(*
		The sequence manager co-ordinates the selection and execution of 
		machine sequences. Machine sequences are created by extending the 
		FB_SequenceBase FB.
*)
FUNCTION_BLOCK FB_SequenceManager_ss
VAR	
	//aSequences: ARRAY[1..5] OF POINTER TO FB_SequenceBase;
	 
	nNumberSequences: INT := 0;
	
	{attribute 'OPC.UA.DA' := '1'} 
	eState:  E_SequenceState := E_SequenceState.STOP; //always stop sequences after PLC restart
	{attribute 'OPC.UA.DA' := '1'} 
	eStateTarget:  E_SequenceState := E_SequenceState.STOP;
	
	eSMState: (STOPPED, STARTING, RUNNING, HOLD) := STOPPED;
	nCurrentStep: INT := 1;
	nCurrentStepPreviousCycle: INT := 1;
	nCurrentSequence: INT := 1;
	nCurrentStepCheck: INT := 1; // use this to iterate over the sequence steps to check if an interlock has rolled back the sequence
	bPauseAcknowledged: BOOL := FALSE;
	
	
	
	{attribute 'OPC.UA.DA' := '0'} 
	fbTONstep: TON;			// these timers are set using the time values stored in each ST_SequenceStep
	{attribute 'OPC.UA.DA' := '0'} 
	fbTONdelay: TON;
	{attribute 'OPC.UA.DA' := '0'} 
	bIsFirstRun: BOOL := TRUE;
	
	i: INT;
	Steps : ARRAY[1..20] OF ST_SequenceStep;
	
	fbCurrentSequence: FB_SequenceBase;
END_VAR

VAR_IN_OUT
	aSequences: ARRAY[1..10] OF FB_SequenceBase;
	//fbCurrentSequence: FB_SequenceBase;
END_VAR

IF bIsFirstRun THEN
	fbTONdelay.PT := T#0S;
	fbTONdelay.IN := TRUE;
	fbTONdelay.PT := T#0S;
	fbTONstep.IN := FALSE;
	bIsFirstRun := FALSE;
	fbCurrentSequence := aSequences[1];
	eSMState := STOPPED;
END_IF


fbTONstep();
fbTONdelay();


CASE eSMState OF
	
	STOPPED:
		// Wait here until a start sequence command is received
		eState := E_SequenceState.STOP;
		
		
	STARTING:
		FOR i := 1 TO fbCurrentSequence.stepsTotal() BY 1 DO
			Steps := fbCurrentSequence.steps();
			Steps[i].Device^.enable();
		END_FOR
	
		nCurrentStepPreviousCycle := nCurrentStep;
		
		// Attempt next step execution 
		IF executeStep(fbCurrentSequence.step(nCurrentStep)) AND nCurrentStep <> fbCurrentSequence.stepsTotal() THEN
			nCurrentStep := nCurrentStep + 1;
		END_IF
		
		
		// Check which sequence step we are up to, set the currentStep indicator to +1 of where we are
		// Interlocks / permissives can cause us to go backwards in steps, therefore we must do this check
		checkCurrentStep();	
		
		IF nCurrentStep < nCurrentStepPreviousCycle THEN  // an interlock has caused the program to roll back in sequence (interlock etc.) - stay in PAUSE state and wait for user acknowledgement
			eSMState := HOLD;
		END_IF
		
			
		IF nCurrentStep = fbCurrentSequence.stepsTotal() THEN  // check if we have completed all of the steps
			eSMState := RUNNING;
		END_IF
		
		eState := E_SequenceState.STARTING;
	
		
		
		
	RUNNING:
		// Sequence is running - just need to check that we are still running, if not, we go to paused
		nCurrentStepPreviousCycle := nCurrentStep;
		checkCurrentStep();
		
		IF nCurrentStep < fbCurrentSequence.stepsTotal() THEN  // something has forced us out of the running state, go to paused and wait for operator to acknowledge
			eSMState := HOLD;
		END_IF
		
		eState := E_SequenceState.RUN;
		
		IF NOT (fbCurrentSequence.step(StepNum := nCurrentStep)^.Device^.getState() = fbCurrentSequence.stepCommand(StepNumber := nCurrentStep)) THEN
			eSMState := STARTING;
		END_IF
		
	HOLD:
		// Do not progress the sequence until the operator has acknowledged that something went wrong
		IF bPauseAcknowledged THEN
			eSMState := STARTING;
			bPauseAcknowledged := FALSE;
		END_IF
		
		eState := E_SequenceState.HOLD;
END_CASE

METHOD acknowledgePause : BOOL
VAR_INPUT
END_VAR
bPauseAcknowledged := TRUE;
END_METHOD

METHOD addSequence : BOOL
VAR_INPUT
	Sequence: FB_SequenceBase;
END_VAR
aSequences[nNumberSequences + 1] := Sequence;
nNumberSequences := nNumberSequences + 1;
END_METHOD

METHOD checkCurrentStep : BOOL
VAR_INPUT
END_VAR

VAR
	currentState: E_DeviceState;
	targetState: E_DeviceState;
END_VAR
nCurrentStepCheck := 1;

WHILE nCurrentStepCheck < (fbCurrentSequence.stepsTotal() + 1) DO
	
	currentState := fbCurrentSequence.stepState(nCurrentStepCheck);
	targetState := fbCurrentSequence.stepCommand(nCurrentStepCheck);

	IF currentState = targetState THEN
		nCurrentStepCheck := nCurrentStepCheck + 1;
	ELSE
		nCurrentStep := nCurrentStepCheck; // step check reveals we are here
		nCurrentStepCheck := fbCurrentSequence.stepsTotal() + 1; // terminate loop as the checking is finished
	END_IF
END_WHILE
END_METHOD

METHOD executeStep : BOOL
VAR_INPUT
	stSequenceStep: POINTER TO ST_SequenceStep;
END_VAR

VAR
	(*eCheckState: E_DeviceState;
	eCheckStateAlternative: E_DeviceState;
	eCheckStateAlternative2: E_DeviceState;
	eCheckCommand: E_DeviceState;
	fbDevice: POINTER TO FB_BaseDevice;
	*)
END_VAR
executeStep := FALSE;
	
// IF fbCurrentSequence.step(StepNum := nCurrentStep)^.Device^.isEnabled()  THEN 
IF (fbCurrentSequence.step(StepNum := nCurrentStep)^.Device^.isEnabled() ) AND 
		(NOT (fbCurrentSequence.step(StepNum := nCurrentStep)^.Device^.getMode() = E_DeviceMode.MANUAL)) THEN 
	//AND fbTONdelay.Q THEN
		
		//fbTONdelay.IN := FALSE; 		
		fbTONstep(IN:= TRUE, PT := stSequenceStep^.StepMinDuration);		
		stSequenceStep^.Device^.setCommand(StateTarget := stSequenceStep^.Command); // set the target state 

END_IF

(*
IF fbCurrentSequence.step(StepNum := nCurrentStep)^.Device^.getState()  
	= fbCurrentSequence.step(StepNum := nCurrentStep)^.Device^.getCommand() 
	AND fbTONstep.Q THEN  *)


IF fbCurrentSequence.step(StepNum := nCurrentStep)^.Device^.getState()  
	= fbCurrentSequence.stepCommand(StepNumber := nCurrentStep)
	AND fbTONstep.Q THEN  
	
	fbTONstep.IN := FALSE; 
	fbTONdelay.IN := FALSE;
	fbTONdelay(IN:= TRUE, PT := stSequenceStep^.DelayUntilNextStep); 
	
	executeStep := TRUE; // indicate that the step was sucessful
	
END_IF
END_METHOD

METHOD getCurrentSeq_FB : POINTER TO FB_SequenceBase
VAR_INPUT
END_VAR
getCurrentSeq_FB := ADR(fbCurrentSequence);
END_METHOD

METHOD getCurrentSeq_ID : INT
VAR_INPUT
END_VAR
getCurrentSeq_ID := nCurrentSequence;
END_METHOD

METHOD getState : E_SequenceState
VAR_INPUT
END_VAR
getState := eState;
END_METHOD

METHOD initSequence : BOOL
VAR_INPUT
END_VAR
// We want to iterate through all of the components in a sequence and enable them.
// We also want to disable any other device (provided it is not in manual)
END_METHOD

METHOD pauseSequence : BOOL
VAR_INPUT
END_VAR
eSMState := HOLD;
END_METHOD

METHOD selectSequence : BOOL
VAR_INPUT
	Sequence: INT;
END_VAR
fbCurrentSequence := aSequences[Sequence];
nCurrentSequence := Sequence;
END_METHOD

METHOD startSequence : BOOL
VAR_INPUT
END_VAR
VAR

END_VAR
eSMState := STARTING;

FOR i := 1 TO fbCurrentSequence.stepsTotal() BY 1 DO
	Steps := fbCurrentSequence.steps();
	Steps[i].Device^.enable();
END_FOR

nCurrentStep := 1;
nCurrentStepPreviousCycle := 1;
//nCurrentSequence := 1;
nCurrentStepCheck := 1;
END_METHOD

METHOD stopSequence : BOOL
VAR_INPUT
END_VAR
eSMState := STOPPED;


FOR i := 1 TO fbCurrentSequence.stepsTotal() BY 1 DO
	Steps := fbCurrentSequence.steps();
	Steps[i].Device^.disable();
END_FOR
END_METHOD

END_FUNCTION_BLOCK

(* stored: Version 1.1.0.1, ProductVersion 3.1.4024.12
   POU FB_SequenceManager_ss: Id {ca4fc9b5-2c45-4a55-b8ba-5233f3330b99}, SpecialFunc None
   Method acknowledgePause: Id {e6cb5dd8-a3f8-4b1a-95f3-e07fb80fc81b}
   Method addSequence: Id {4f9f888e-316b-4ee7-af47-7abc95aa55d8}
   Method checkCurrentStep: Id {77646001-508b-4614-ab8f-0db1d6059483}
   Method executeStep: Id {7cb1c551-5162-49d1-b9d2-4f0e1594d359}
   Method getCurrentSeq_FB: Id {ebe0a736-cfec-4877-8022-f0159ebcaf12}
   Method getCurrentSeq_ID: Id {45465c3a-30d1-4276-8734-985f502a8975}
   Method getState: Id {148368fe-5d27-4d73-8a28-303eb0cdfe1e}
   Method initSequence: Id {4127f791-0f1c-47ff-9217-cf05d8acbbbf}
   Method pauseSequence: Id {39b74db0-72f7-4c7e-8a09-9b4fda077a1d}
   Method selectSequence: Id {89040f6a-d7e0-4b4a-8050-b8f328bba8ae}
   Method startSequence: Id {af996820-e89c-4eaa-9e11-0c9f565d4d3f}
   Method stopSequence: Id {f043cee9-47a6-4b01-960d-aa0e1397f836} *)
